Staubli VAL3: setSignal.pgx

program setSignal(bool x_bCondition (dimensions=1), dio x_doSignal (dimensions=1))
begin
  if x_bCondition
    if !x_doSignal
      x_doSignal=true
    endIf
  endIf
end
